FUNCTION_BLOCK FB_Add
VAR
    refValue : REFERENCE TO INT;
END_VAR

METHOD EXECUTE 
VAR_INPUT
END_VAR
IF refValue <> 0 THEN
    refValue := refValue + 10;
END_IF
END_METHOD

METHOD SetReference 
VAR_INPUT
    iRef : REFERENCE TO INT;
END_VAR
refValue REF= iRef;
END_METHOD

END_FUNCTION_BLOCK

(* stored: Version 1.1.0.1, ProductVersion 3.1.4024.16
   POU FB_Add: Id {41f68d66-c189-4ebc-98ce-b4a42573dec1}, SpecialFunc None
   Method EXECUTE: Id {81726d5a-c0f0-40ec-b8d5-2d185edd3553}
   Method SetReference: Id {464aa2f3-dfbd-4ac0-bc95-24018e26db2d} *)
